{attribute 'linkalways'} 
{attribute 'no_explicit_call' := 'This FB is a CLASS and must be accessed using methods or properties'}
{attribute 'enable_dynamic_creation'}
FUNCTION_BLOCK FINAL MIN_LREAL EXTENDS Node
VAR
	in1 : _LREAL(0.0);
	in2 : _LREAL(0.0);
	out : _LREAL(0.0);
END_VAR

METHOD PUBLIC Clone : I_Node
VAR
	pNode : POINTER TO MIN_LREAL;
END_VAR
pNode := __NEW(MIN_LREAL);
Clone := pNode^;
END_METHOD

METHOD FB_init : BOOL
VAR_INPUT
	bInitRetains : BOOL; // if TRUE, the retain variables are initialized (warm start / cold start)
	bInCopyCode : BOOL;  // if TRUE, the instance afterwards gets moved into the copy code (online change)
END_VAR
AddInput('in1',THIS^.in1);
AddInput('in2',THIS^.in2);
AddOutput('out', THIS^.out);
END_METHOD

METHOD PROTECTED OnExecute
VAR
END_VAR
out.Value := MIN(in1.Value, in2.Value);
END_METHOD

END_FUNCTION_BLOCK

(* stored: Version 1.1.0.1, ProductVersion 3.1.4024.15
   POU MIN_LREAL: Id {6c551d8a-4b6f-4285-85c1-f0bc98b31b0f}, SpecialFunc None
   Folder Constructor: Id {7bba2272-26dd-43e7-bf99-a92932f5e2bd}
   Method Clone: Id {dc196beb-c480-4101-8eca-746d81237776}
   Method FB_init: Id {f2ae3752-19a5-4a78-acf2-32e5849dfa34}
   Method OnExecute: Id {89df5e4a-0061-4635-aad1-a3f852cf70c7} *)
